(* IEC 61131-3 sources: Industry-PLC-LLM/data/PLCBEAD_repo/PLCBEAD_PLCEmbed-main/PLC-BEAD/Source/GEB/FILTER_DW, 1 file *)

(* ---- FILTER_DW.ST ---- *)
FUNCTION_BLOCK T_PLC_MS_block
	VAR_OUTPUT
		T_PLC_MS :	UDINT;
	END_VAR

	VAR
		PLC_TICKS_PER_SEC :	INT;
		PLC_SYS_TICK_CNT :	DINT;
	END_VAR

	VAR
		debug :	BOOL;(*Debug-Mode ON / OFF*)
		N :	INT;(*Debug-Faktor*)
		Offset :	UDINT;(*Debug-Offset*)
		temp :	DWORD := DWORD#1;(*Debug-Offset*)
		MODE :	BOOL;(*modus*)
		faktor :	UDINT;(*Systemtakt-Faktor*)
		init :	BOOL;
		v_plc_ticks_per_sec :	UDINT;
		base :	UDINT := UDINT#1000;
	END_VAR

	IF init = FALSE THEN
		v_plc_ticks_per_sec := INT_TO_UDINT(PLC_TICKS_PER_SEC);
		IF v_plc_ticks_per_sec = UDINT#1024 THEN
			faktor := UDINT#1;
			MODE := FALSE;
		ELSIF v_plc_ticks_per_sec > UDINT#0 THEN
			IF v_plc_ticks_per_sec <= base THEN
				faktor := base / v_plc_ticks_per_sec;
				MODE := FALSE;
			ELSE
				faktor := v_plc_ticks_per_sec / base;
				MODE := TRUE;
			END_IF;
		ELSE
			faktor := UDINT#1;
		END_IF;
		init := TRUE;
	END_IF;

	IF MODE THEN
		T_PLC_MS := DINT_TO_UDINT(PLC_SYS_TICK_CNT) / faktor;
	ELSE
		T_PLC_MS := DINT_TO_UDINT(PLC_SYS_TICK_CNT) * faktor;
	END_IF;

	IF debug THEN
		T_PLC_MS := (DWORD_TO_UDINT(SHL(UDINT_TO_DWORD(T_PLC_MS),N) OR SHL(temp,N)) - UDINT#1) + Offset;
	END_IF;

END_FUNCTION_BLOCK

FUNCTION _DWORD_TO_REAL:REAL
	VAR_INPUT
		IN :	DWORD;
	END_VAR

	_DWORD_TO_REAL := UDINT_TO_REAL(DWORD_TO_UDINT(IN));
END_FUNCTION

FUNCTION _REAL_TO_DWORD: DWORD

  VAR_INPUT
    X :	REAL;
  END_VAR

  IF REAL_TO_DWORD(0.5) = DWORD#1 THEN
    _REAL_TO_DWORD := REAL_TO_DWORD(X);
  ELSIF X > 0.0 THEN
    _REAL_TO_DWORD := REAL_TO_DWORD(X+0.5);
  ELSIF X < 0.0 THEN
    _REAL_TO_DWORD := REAL_TO_DWORD(X-0.5);
  ELSE
    _REAL_TO_DWORD := DWORD#0;
  END_IF;
END_FUNCTION

FUNCTION_BLOCK FILTER_DW

	VAR_INPUT
		X :	DWORD;
		T :	TIME;
	END_VAR

	VAR_OUTPUT
		Y :	DWORD;
	END_VAR

	VAR
		last :	UDINT;
		TX :	UDINT;
		init :	BOOL;
		Yi :	REAL;
		T_PLC_MS :	T_PLC_MS_block;
	END_VAR

	T_PLC_MS();
	TX:= T_PLC_MS.T_PLC_MS;

	IF NOT init OR T = t#0s THEN
		init := TRUE;
		Yi := _DWORD_TO_REAL(X);
	ELSE
		Yi := Yi + (_DWORD_TO_REAL(X) - _DWORD_TO_REAL(Y)) * UDINT_TO_REAL(TX - last) / TIME_TO_REAL(T);
	END_IF;
	last := TX;

	Y := _REAL_TO_DWORD(Yi);

END_FUNCTION_BLOCK

PROGRAM program0
  VAR
	X :	DWORD;
	T :	TIME;

	Y :	DWORD;

	func_block : FILTER_DW;
  END_VAR
	func_block.X  := X;
	func_block.T  := T;
	func_block();
	Y := func_block.Y;
END_PROGRAM
